# B&R Automation Studio project Lektion_12_agdp
Automation Studio 4.8.2.72

## Configuration Config1

### Task classes (Cpu.sw)
```
Cyclic#1:
  Program <- Program.prg
  Program1 <- Program1.prg
Cyclic#5:
  Program2 <- Program2.prg
  Program3 <- Program3.prg
Cyclic#6:
  Program4 <- Program4.prg
Binaries: udbdef, FWRules, TCData, sysconf, Role, User, iomap, ashwd, asfw, arconfig, ashwac
Libraries: runtime, astime, asieccon
```

### Hardware
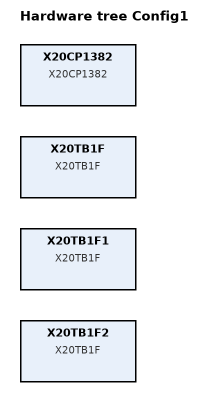
```
X20CP1382 : X20CP1382 v1.10.0.0  [X1 -> X1.SL; X2 -> X2.SL; X3 -> X3.SL]
  Module X1 (Type=X1, Virtual=true, Version=1.10.0.0)
    Connection (Connector=SS1, TargetModule=X20TB1F, TargetConnector=SS)
    Connection (Connector=SL, TargetModule=X20CP1382, TargetConnector=X1)
  Module X2 (Type=X2, Virtual=true, Version=1.10.0.0)
    Connection (Connector=SS1, TargetModule=X20TB1F1, TargetConnector=SS)
    Connection (Connector=SL, TargetModule=X20CP1382, TargetConnector=X2)
  Module X3 (Type=X3, Virtual=true, Version=1.10.0.0)
    Connection (Connector=SS1, TargetModule=X20TB1F2, TargetConnector=SS)
    Connection (Connector=SL, TargetModule=X20CP1382, TargetConnector=X3)
  Connector IF2:
    ActivateDevice = 1
  ConfigurationID = Lektion_12_agdp_Config1
  Simulation = 1
X20TB1F : X20TB1F v1.0.0.0
X20TB1F1 : X20TB1F v1.0.0.0
X20TB1F2 : X20TB1F v1.0.0.0
```

## Logical view

### Program Logical/Program (IEC)

#### Main.st - Init, cyclic, exit code
```iecst
PROGRAM _INIT
	(* Insert code here *)
	a := 4.0;
	b := 3.0;
END_PROGRAM

PROGRAM _CYCLIC
	(* Insert code here *)

	c := PYTHA(a, b);

END_PROGRAM

PROGRAM _EXIT
	(* Insert code here *)

END_PROGRAM
```

#### Variables.var - Local variables
```iecst
VAR
	c : LREAL;
	b : REAL;
	a : REAL;
END_VAR
```

#### LocalFunctions.fun
```iecst
{REDUND_ERROR} FUNCTION PYTHA : LREAL (*TODO: Add your comment here*) (*$GROUP=User,$CAT=User,$GROUPICON=User.png,$CATICON=User.png*)
	VAR_INPUT
		a : REAL;
		b : REAL;
	END_VAR
END_FUNCTION
```

#### PYTHA.st
```iecst
(* TODO: Add your comment here *)
FUNCTION PYTHA

	PYTHA := SQRT(a**2 + b**2);

END_FUNCTION
```

### Program Logical/Program1 (IEC)

#### Main.st - Init, cyclic, exit code
```iecst
PROGRAM _INIT
	(* Insert code here *)
	A := TRUE;
	B := TRUE;
	C := TRUE;

END_PROGRAM

PROGRAM _CYCLIC
	(* Insert code here *)

	output := FUCKR(A, B, C);

END_PROGRAM

PROGRAM _EXIT
	(* Insert code here *)

END_PROGRAM
```

#### Variables.var - Local variables
```iecst
VAR
	B : BOOL;
	C : BOOL;
	A : BOOL;
	output : BOOL;
END_VAR
```

#### LocalFunctions.fun
```iecst
{REDUND_ERROR} FUNCTION FUCKR : BOOL (*TODO: Add your comment here*) (*$GROUP=User,$CAT=User,$GROUPICON=User.png,$CATICON=User.png*)
	VAR_INPUT
		A : BOOL;
		B : BOOL;
		C : BOOL;
	END_VAR
END_FUNCTION
```

#### FUCKR.st
```iecst
(* TODO: Add your comment here *)
FUNCTION FUCKR

	FUCKR := (NOT(A) AND B AND C) OR (A AND NOT(B) AND C) OR (A AND B AND NOT(C)) OR (A AND B AND C);

END_FUNCTION
```

### Program Logical/Program2 (IEC)

#### Main.st - Init, cyclic, exit code
```iecst
PROGRAM _INIT
	(* Insert code here *)
	 input := FALSE;
END_PROGRAM

PROGRAM _CYCLIC
	(* Insert code here *)
	r_trigger(in := input);
	output := r_trigger.Q;

END_PROGRAM

PROGRAM _EXIT
	(* Insert code here *)

END_PROGRAM
```

#### Variables.var - Local variables
```iecst
VAR
	output : BOOL;
	input : BOOL;
END_VAR
VAR RETAIN
	r_trigger : R_EDGETRIG;
END_VAR
```

#### LocalFunctions.fun
```iecst
{REDUND_ERROR} FUNCTION_BLOCK R_EDGETRIG (*TODO: Add your comment here*) (*$GROUP=User,$CAT=User,$GROUPICON=User.png,$CATICON=User.png*)
	VAR_INPUT
		in : BOOL;
	END_VAR
	VAR_OUTPUT
		Q : BOOL;
	END_VAR
	VAR RETAIN
		old_in : BOOL;
	END_VAR
END_FUNCTION_BLOCK
```

#### R_EDGETRIG.st
```iecst
(* TODO: Add your comment here *)
FUNCTION_BLOCK R_EDGETRIG

	Q := NOT old_in AND in;
	old_in := in;

END_FUNCTION_BLOCK
```

### Program Logical/Program3 (IEC)

#### Variables.var
```iecst
VAR
	output : BOOL;
	input : BOOL;
END_VAR
VAR RETAIN
	r_trigger : RF_EDGETRIG;
END_VAR
```

#### LocalFunctions.fun
```iecst
{REDUND_ERROR} FUNCTION_BLOCK RF_EDGETRIG (*TODO: Add your comment here*) (*$GROUP=User,$CAT=User,$GROUPICON=User.png,$CATICON=User.png*)
	VAR_INPUT
		in : BOOL;
	END_VAR
	VAR_OUTPUT
		Q : BOOL;
	END_VAR
	VAR RETAIN
		old_in : BOOL;
	END_VAR
END_FUNCTION_BLOCK
```

#### R_EDGETRIG.st
```iecst
(* TODO: Add your comment here *)
FUNCTION_BLOCK RF_EDGETRIG

	Q := (NOT old_in AND in) OR (old_in AND NOT in);
	old_in := in;

END_FUNCTION_BLOCK
```

### Program Logical/Program4 (IEC)

#### Main.st - Init, cyclic, exit code
```iecst
PROGRAM _INIT
	(* Insert code here *)
	enable := TRUE;
	next_state := FALSE;
END_PROGRAM

PROGRAM _CYCLIC
	(* Insert code here *)

	state_machine(EN := enable, NS := next_state);
	state := state_machine.Q;
END_PROGRAM

PROGRAM _EXIT
	(* Insert code here *)

END_PROGRAM
```

#### Types.typ - Local data types
```iecst
TYPE
	STATES :
		(
		STOP,
		STARTING,
		EXECUTE,
		COMPLETE,
		RESETTING
		);
END_TYPE
```

#### Variables.var - Local variables
```iecst
VAR
	state_machine : STATE_MACHINE;
	next_state : BOOL;
	state : STATES;
	enable : BOOL;
END_VAR
```

#### LocalFunctions.fun
```iecst
{REDUND_ERROR} FUNCTION_BLOCK STATE_MACHINE (*TODO: Add your comment here*) (*$GROUP=User,$CAT=User,$GROUPICON=User.png,$CATICON=User.png*)
	VAR_INPUT
		EN : BOOL;
		NS : BOOL;
	END_VAR
	VAR_OUTPUT
		Q : STATES;
		ERR : BOOL;
	END_VAR
END_FUNCTION_BLOCK
```

#### STATE_MACHINE.st
```iecst
(* TODO: Add your comment here *)
FUNCTION_BLOCK STATE_MACHINE

	CASE Q OF
		STOP:
			IF EN THEN
				Q := STARTING;
			END_IF;
		STARTING:
			IF NOT EN THEN
				Q := STOP;
			ELSE
				IF NS THEN
					Q := EXECUTE;
				END_IF;
			END_IF;
		EXECUTE:
			IF NOT EN THEN
				Q := STOP;
			ELSE
				IF NS THEN
	  				Q := COMPLETE;
				END_IF;
			END_IF;

		COMPLETE:
			IF NOT EN THEN
				Q := STOP;
			ELSE
				IF NS THEN
					Q := RESETTING;
				END_IF;
			END_IF;

		RESETTING:
			IF NOT EN THEN
				Q := STOP;
			ELSE
				IF NS THEN
					Q := STARTING;
				END_IF;
			END_IF;

	END_CASE;

END_FUNCTION_BLOCK
```

Listed in the project but not available here: Logical/Global.typ, Logical/Global.var, Logical/Libraries, Logical/Program/Types.typ, Logical/Program1/Types.typ, Logical/Program2/Types.typ
